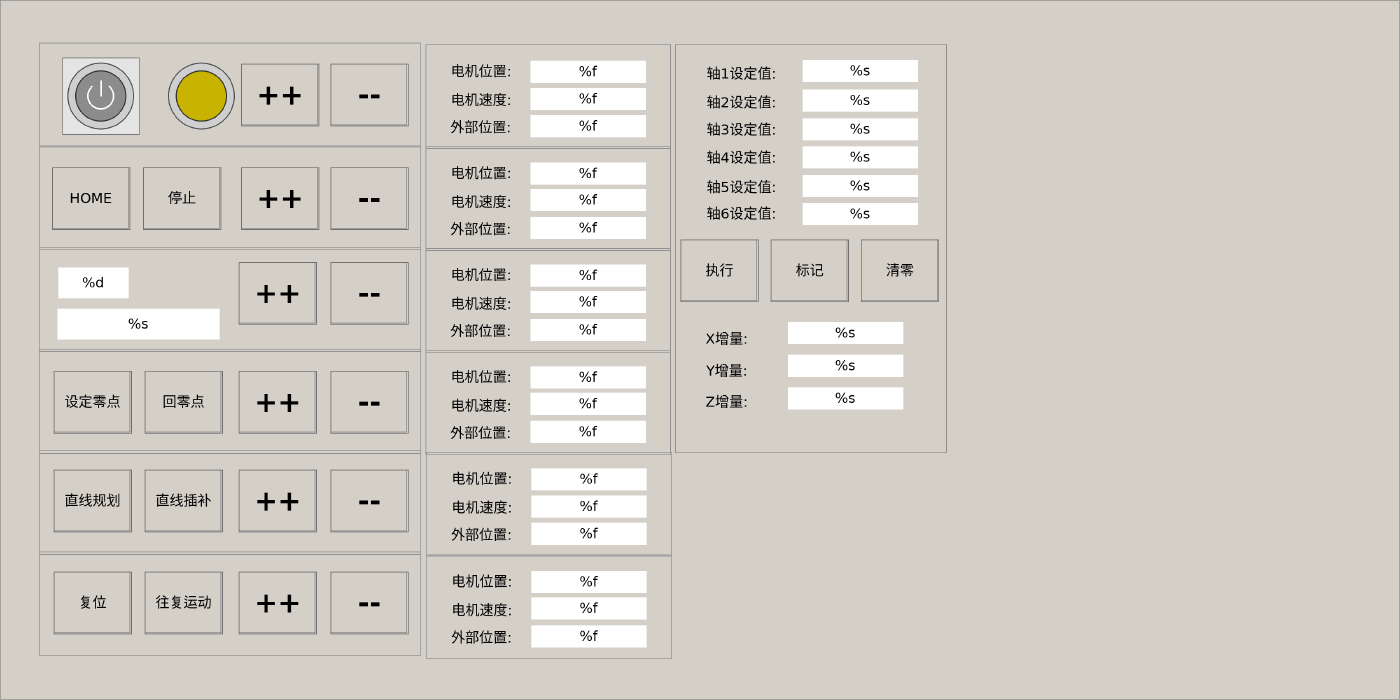
VISUALIZATION Visualization  // 1800x900
    GroupBox (50,47 491x142)
        Button (375,35 100x80), "--"
            OnMouseDown: execute { axisNum:=0; MAIN.CurrentJob:=4; }
            OnMouseUp: execute { axisNum:=0; MAIN.CurrentJob:=0; }
        Button (260,35 100x80), "++"
            OnMouseDown: execute { axisNum:=0; MAIN.CurrentJob:=3; }
            OnMouseUp: execute { axisNum:=0; MAIN.CurrentJob:=0; }
        PowerSwitch (17,27 125x99), variable: MAIN.POWER, behaviour: TOGGLE, style: Switch-PowerSwitch-Gray
        Lamp1 (134,27 150x99), variable: MAIN.LAMP, style: Lamp-Lamp1-Yellow
    GroupBox (547,49 315x142)
        Label (2,28 139x30), "电机位置:"
        Label (4,100 134x30), "外部位置:"
        Textfield (134,63 150x30), "%f", text variable: Axis[0].NcToPlc.ActVelo
        Textfield (134,28 150x30), "%f", text variable: Axis[0].NcToPlc.ActPos
        Textfield (134,98 150x30), "%f", text variable: ExtPos[0]
        Label (9,65 125x30), "电机速度:"
    GroupBox (547,180 315x142)
        Label (2,28 139x30), "电机位置:"
        Label (4,100 134x30), "外部位置:"
        Textfield (134,62 150x30), "%f", text variable: Axis[1].NcToPlc.ActVelo
        Textfield (134,28 150x30), "%f", text variable: Axis[1].NcToPlc.ActPos
        Textfield (134,98 150x30), "%f", text variable: ExtPos[1]
        Label (9,65 125x30), "电机速度:"
    GroupBox (547,311 315x142)
        Label (2,28 139x30), "电机位置:"
        Label (4,100 134x30), "外部位置:"
        Textfield (134,62 150x30), "%f", text variable: Axis[2].NcToPlc.ActVelo
        Textfield (134,28 150x30), "%f", text variable: Axis[2].NcToPlc.ActPos
        Textfield (134,98 150x30), "%f", text variable: ExtPos[2]
        Label (9,65 125x30), "电机速度:"
    GroupBox (547,442 315x142)
        Label (2,28 139x30), "电机位置:"
        Label (4,100 134x30), "外部位置:"
        Textfield (134,62 150x30), "%f", text variable: Axis[3].NcToPlc.ActVelo
        Textfield (134,28 150x30), "%f", text variable: Axis[3].NcToPlc.ActPos
        Textfield (134,98 150x30), "%f", text variable: ExtPos[3]
        Label (9,65 125x30), "电机速度:"
    GroupBox (548,573 315x142)
        Label (2,28 139x30), "电机位置:"
        Label (4,100 134x30), "外部位置:"
        Textfield (134,63 150x30), "%f", text variable: Axis[4].NcToPlc.ActVelo
        Textfield (134,28 150x30), "%f", text variable: Axis[4].NcToPlc.ActPos
        Textfield (134,98 150x30), "%f", text variable: ExtPos[4]
        Label (9,65 125x30), "电机速度:"
    GroupBox (50,179 491x142)
        Button (260,36 100x80), "++"
            OnMouseDown: execute { axisNum:=1; MAIN.CurrentJob:=3; }
            OnMouseUp: execute { axisNum:=1; MAIN.CurrentJob:=0; }
        Button (375,36 100x80), "--"
            OnMouseDown: execute { axisNum:=1; MAIN.CurrentJob:=4; }
            OnMouseUp: execute { axisNum:=1; MAIN.CurrentJob:=0; }
        Button (134,36 100x80), "停止"
            OnMouseClick: execute { MAIN.CurrentJob:=5; }
        Button (17,36 100x80), "HOME"
            OnMouseClick: execute { MAIN.CurrentJob:=6; }
    GroupBox (548,705 315x142)
        Label (2,28 139x30), "电机位置:"
        Label (4,100 134x30), "外部位置:"
        Textfield (134,62 150x30), "%f", text variable: Axis[5].NcToPlc.ActVelo
        Textfield (134,28 150x30), "%f", text variable: Axis[5].NcToPlc.ActPos
        Textfield (134,98 150x30), "%f", text variable: ExtPos[5]
        Label (9,65 125x30), "电机速度:"
    GroupBox (50,310 491x142)
        Button (257,27 100x80), "++"
            OnMouseDown: execute { axisNum:=2; MAIN.CurrentJob:=3; }
            OnMouseUp: execute { axisNum:=2; MAIN.CurrentJob:=0; }
        Button (375,27 100x80), "--"
            OnMouseDown: execute { axisNum:=2; MAIN.CurrentJob:=4; }
            OnMouseUp: execute { axisNum:=2; MAIN.CurrentJob:=0; }
        Textfield (24,33 92x41), "%d", text variable: MAIN.CurrentJob
        Textfield (23,86 210x41), "%s", text variable: MAIN.CurrentJobState
    GroupBox (50,441 491x142)
        Button (257,36 100x80), "++"
            OnMouseDown: execute { axisNum:=3; MAIN.CurrentJob:=3; }
            OnMouseUp: execute { axisNum:=3; MAIN.CurrentJob:=0; }
        Button (375,36 100x80), "--"
            OnMouseDown: execute { axisNum:=3; MAIN.CurrentJob:=4; }
            OnMouseUp: execute { axisNum:=3; MAIN.CurrentJob:=0; }
        Button (19,36 100x80), "设定零点"
            OnMouseClick: execute { MAIN.CurrentJob:=1; }
        Button (136,36 100x80), "回零点"
            OnMouseClick: execute { MAIN.CurrentJob:=11; }
    GroupBox (50,571 491x142)
        Button (257,33 100x80), "++"
            OnMouseDown: execute { axisNum:=4; MAIN.CurrentJob:=3; }
            OnMouseUp: execute { axisNum:=4; MAIN.CurrentJob:=0; }
        Button (375,33 100x80), "--"
            OnMouseDown: execute { axisNum:=4; MAIN.CurrentJob:=4; }
            OnMouseUp: execute { axisNum:=4; MAIN.CurrentJob:=0; }
        Button (19,33 100x80), "直线规划"
            OnMouseClick: execute { MAIN.CurrentJob:=10; }
        Button (136,33 100x80), "直线插补"
            OnMouseClick: execute { MAIN.CurrentJob:=2; }
    GroupBox (50,701 491x142)
        Button (257,34 100x80), "++"
            OnMouseDown: execute { axisNum:=5; MAIN.CurrentJob:=3; }
            OnMouseUp: execute { axisNum:=5; MAIN.CurrentJob:=0; }
        Button (375,34 100x80), "--"
            OnMouseDown: execute { axisNum:=5; MAIN.CurrentJob:=4; }
            OnMouseUp: execute { axisNum:=5; MAIN.CurrentJob:=0; }
        Button (19,34 100x80), "复位"
            OnMouseClick: execute {
                MAIN.CurrentJob:=9;
                //MoveA[0]:=-743179.666443;
                //MoveA[1]:=1499.826050;
                //MoveA[2]:=-1396.145325;
                //MoveA[3]:=6061.5802;
                //MoveA[4]:=1828.031616;
                //MoveA[5]:=-1145.742188;
            }
        Button (136,34 100x80), "往复运动"
            OnMouseClick: execute { MAIN.CurrentJob:=8; }
    GroupBox (868,49 349x533)
        Textfield (163,27 150x30), "%s", text variable: GVL.MoveAString[0]
            OnMouseClick: write MoveAString[0] via Edit
        Textfield (163,65 150x30), "%s", text variable: GVL.MoveAString[1]
            OnMouseClick: write MoveAString[1] via Edit
        Textfield (163,102 150x30), "%s", text variable: GVL.MoveAString[2]
            OnMouseClick: write MoveAString[2] via Edit
        Textfield (163,138 150x30), "%s", text variable: GVL.MoveAString[3]
            OnMouseClick: write MoveAString[3] via Edit
        Textfield (163,175 150x30), "%s", text variable: GVL.MoveAString[4]
            OnMouseClick: write MoveAString[4] via Edit
        Textfield (163,211 150x30), "%s", text variable: GVL.MoveAString[5]
            OnMouseClick: write MoveAString[5] via Edit
        Label (16,31 139x30), "轴1设定值:"
        Label (16,68 139x30), "轴2设定值:"
        Label (16,103 139x30), "轴3设定值:"
        Label (16,139 139x30), "轴4设定值:"
        Label (16,177 139x30), "轴5设定值:"
        Label (16,211 139x30), "轴6设定值:"
        Button (7,259 100x80), "执行"
            OnMouseClick: execute { MAIN.CurrentJob:=7; }
        Button (123,259 100x80), "标记"
            OnMouseClick: execute {
                MoveA[0]:=Axis[0].NcToPlc.ActPos;
                MoveA[1]:=Axis[1].NcToPlc.ActPos;
                MoveA[2]:=Axis[2].NcToPlc.ActPos;
                MoveA[3]:=Axis[3].NcToPlc.ActPos;
                MoveA[4]:=Axis[4].NcToPlc.ActPos;
                MoveA[5]:=Axis[5].NcToPlc.ActPos;
                MoveAString[0]:=LREAL_TO_STRING(MoveA[0]/24.995);
                MoveAString[1]:=LREAL_TO_STRING(MoveA[1]/32.28);
                MoveAString[2]:=LREAL_TO_STRING(MoveA[2]/49.845);
                MoveAString[3]:=LREAL_TO_STRING(MoveA[3]/50.905);
                MoveAString[4]:=LREAL_TO_STRING(MoveA[4]/80.34);
                MoveAString[5]:=LREAL_TO_STRING(MoveA[5]/60.5);
            }
        Button (239,259 100x80), "清零"
            OnMouseClick: execute {
                MoveA[0]:=0;
                MoveA[1]:=0;
                MoveA[2]:=0;
                MoveA[3]:=0;
                MoveA[4]:=0;
                MoveA[5]:=0;
                MoveAString[0]:='0';
                MoveAString[1]:='0';
                MoveAString[2]:='0';
                MoveAString[3]:='0';
                MoveAString[4]:='0';
                MoveAString[5]:='0';
            }
        Textfield (144,364 150x30), "%s", text variable: GVL.OutMovePosString[0]
            OnMouseClick: write OutMovePosString[0] via Edit
        Textfield (144,406 150x30), "%s", text variable: GVL.OutMovePosString[1]
            OnMouseClick: write OutMovePosString[1] via Edit
        Textfield (144,448 150x30), "%s", text variable: GVL.OutMovePosString[2]
            OnMouseClick: write OutMovePosString[2] via Edit
    Label (865,421 139x30), "X增量:"
    Label (865,462 139x30), "Y增量:"
    Label (865,502 139x30), "Z增量:"
END_VISUALIZATION

(* stored: Version 1.1.0.1, ProductVersion 3.1.4018.5
   Visu Visualization: Id {4b3000ae-8bfc-4343-82c7-89025f75f23c} *)
